// Mitsubishi GX Works2 project: Exercicio semaforo   PLC: Q03UDV

PROGRAM MAIN
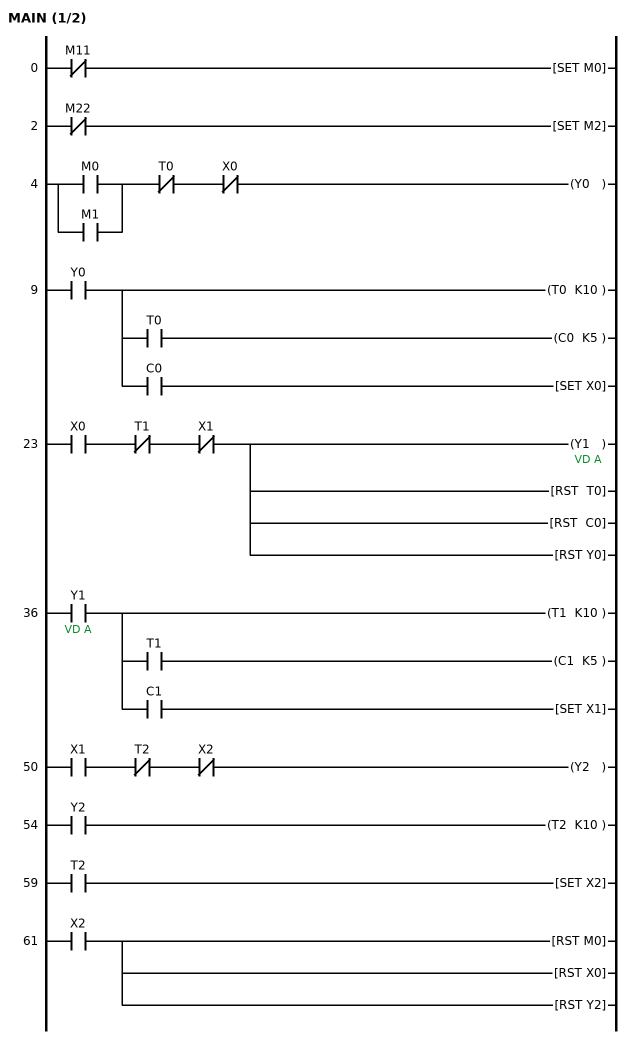
0     LDI     M11
      SET     M0
2     LDI     M22
      SET     M2
4     LD      M0
      OR      M1
      ANI     T0
      ANI     X0
      OUT     Y0
9     LD      Y0
      OUT     T0 K10
      MPS
      AND     T0
      OUT     C0 K5
      MPP
      AND     C0
      SET     X0
23    LD      X0
      ANI     T1
      ANI     X1
      OUT     Y1  ; VD A
      RST     T0
      RST     C0
      RST     Y0
36    LD      Y1  ; VD A
      OUT     T1 K10
      MPS
      AND     T1
      OUT     C1 K5
      MPP
      AND     C1
      SET     X1
50    LD      X1
      ANI     T2
      ANI     X2
      OUT     Y2
54    LD      Y2
      OUT     T2 K10
59    LD      T2
      SET     X2
61    LD      X2
      RST     M0
      RST     X0
      RST     Y2
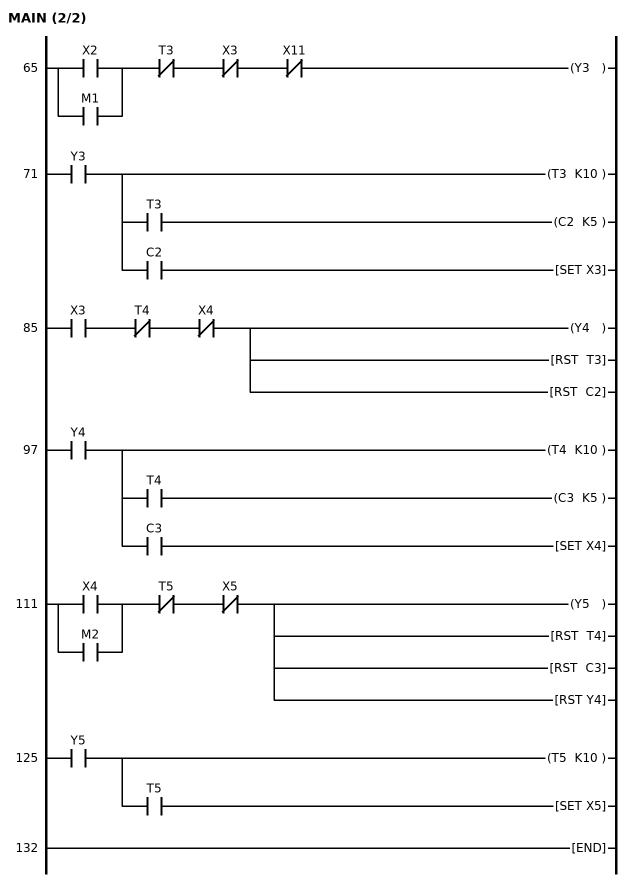
65    LD      X2
      OR      M1
      ANI     T3
      ANI     X3
      ANI     X11
      OUT     Y3
71    LD      Y3
      OUT     T3 K10
      MPS
      AND     T3
      OUT     C2 K5
      MPP
      AND     C2
      SET     X3
85    LD      X3
      ANI     T4
      ANI     X4
      OUT     Y4
      RST     T3
      RST     C2
97    LD      Y4
      OUT     T4 K10
      MPS
      AND     T4
      OUT     C3 K5
      MPP
      AND     C3
      SET     X4
111   LD      X4
      OR      M2
      ANI     T5
      ANI     X5
      OUT     Y5
      RST     T4
      RST     C3
      RST     Y4
125   LD      Y5
      OUT     T5 K10
      AND     T5
      SET     X5
132   END
END_PROGRAM
